TYPE ST_HMI_DataSourceHist : 
STRUCT
	nCurrentRecordID: DINT;
	stSourceInfo: ST_HMI_DataSourceHistInfo;
	nRecordCount: DINT;
	aRecords: ARRAY [0..255] OF ST_HMI_DataSourceHistRecordInfo;
END_STRUCT
END_TYPE

(* stored: DUT ST_HMI_DataSourceHist: Id 0bce22b0-74b0-4773-9b13-8c4b20751dbf *)
